{attribute 'qualified_only'}
VAR_GLOBAL
	Logger	: ZigaLibs_Logging.FB_Logger;
END_VAR

(* stored: Version 1.1.0.1, ProductVersion 3.1.4024.13
   GVL GVL_Bronkhorst: Id {76cb8281-5d0d-05db-328e-6cb5b830da61} *)
